FUNCTION_BLOCK MECH1_DIAGL (* Diagnostic for a Unidirectional Mechanism with local Clocking and Publication *)
  (* Standard: 61499-1; Classification: Diagnostics; ApplicationDomain: Mechanisms *)
  (* Version 0.1, 2004-10-20, JHC, Rockwell Automation, Renamed to replace old MECH1_DIAGL. *)
  (* Version 0.0, 2004-09-26, JHC, Rockwell Automation, Derived from MECH2_DIAG; made composite, incorporated clock. *)
  (* Compiler header: package fb.rt.mva; import fb.rt.net.*; *)
  (* Compiler Java Sun JDK 1.4.2 *)
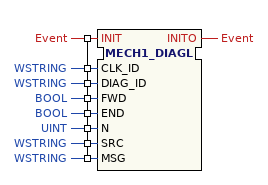
  EVENT_INPUT
    INIT WITH CLK_ID, DIAG_ID, N, SRC, MSG, END, FWD, N;
  END_EVENT
  EVENT_OUTPUT
    INITO;
  END_EVENT
  VAR_INPUT
    CLK_ID : WSTRING := "DIAG_CLK"; (* Diagnostic Clock Local Channel ID *)
    DIAG_ID : WSTRING := "DIAG"; (* Diagnostic output channel ID *)
    FWD : BOOL; (* Forward Actuation Command from Controller *)
    END : BOOL; (* END(Fully Advanced)Sensor *)
    N : UINT; (* Timeout Period in CLK cycles *)
    SRC : WSTRING; (* Diagnostic Source ID *)
    MSG : WSTRING := "TIMEOUT_ADVANCING"; (* Fault message *)
  END_VAR
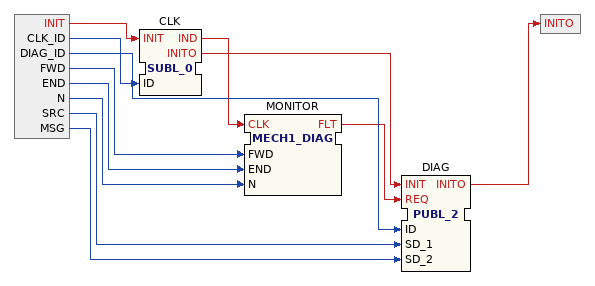
  FBS
    MONITOR : MECH1_DIAG;
    CLK : SUBL_0;
    DIAG : PUBL_2;
  END_FBS
  EVENT_CONNECTIONS
    INIT TO CLK.INIT;
    CLK.IND TO MONITOR.CLK;
    CLK.INITO TO DIAG.INIT;
    MONITOR.FLT TO DIAG.REQ;
    DIAG.INITO TO INITO;
  END_CONNECTIONS
  DATA_CONNECTIONS
    DIAG_ID TO DIAG.ID;
    SRC TO DIAG.SD_1;
    MSG TO DIAG.SD_2;
    CLK_ID TO CLK.ID;
    FWD TO MONITOR.FWD;
    END TO MONITOR.END;
    N TO MONITOR.N;
  END_CONNECTIONS
END_FUNCTION_BLOCK
